// TIA Portal V20 export
// export: Created 2025-12-01T14:56:28.7894761Z, ExportSetting None, DisplayName Totally Integrated Automation Portal, DisplayVersion V20 Update 3, DisplayName TIA Portal Openness, DisplayVersion V20 Update 3, DisplayName TIA Portal Version Control Interface, DisplayVersion V20 Update 3, DisplayName STEP 7 Professional, DisplayVersion V20 Update 3, DisplayName STEP 7 Safety, DisplayVersion V20 Update 2, DisplayName WinCC Basic/Comfort/Advanced, DisplayVersion V20 Update 3, DisplayName WinCC Professional, DisplayVersion V20 Update 3, DisplayName WinCC Unified, DisplayVersion V20 Update 3
FUNCTION_BLOCK "FB415_EST_Girador_180G"   // FB415, LAD
TITLE = Control del Ramal de Salidas
{ S7_Optimized_Access := 'FALSE' }
AUTHOR : TLigero
NAME : 20160208
VERSION : 3.2
// FECHA:    27/05/2014  AUTOR: N.Rodriguez
// INSTALACION: Santomera Ampliacion 2FSS
// //////////////////////////////////
// // Registro Incidencias   ////////
// //////////////////////////////////
// FECHA:   AUTOR MODIFICACION: 
// DESCRIPCION:
// stored: AutoNumber false, SetENOAutomatically false
   VAR_INPUT
      Mesa : UInt;
      En_Tension : Bool;
      pHs_Tope : Bool;
      In_Tope_Up : Bool;
      In_Tope_Dw : Bool;
      In_Gir_Pos0 : Bool;
      In_Gir_Pos180 : Bool;
      In_Gir_Up : Bool;
      In_Gir_Dw : Bool;
      Termico_E1S3 : Bool;
      Avance_E1S3 : Bool;
      NXT_CargaOK : Bool;
      NXT_Avance : Bool;
      PRV_AVTF : Bool;
      V_TMPAus_Salida : UDInt;
      V_TMPVaciado : Time := T#10S;
      V_TOUT_Avance : Time := T#15S;
      V_TOUT_Giro_Girador : Time := T#5S;
      V_TOUT_Tope : Time := T#5S;
      V_TOUT_Elevacion_Girador : Time;
      V_TMP_Centrado : Time;
   END_VAR
   VAR_OUTPUT
      PRV_CARGA_OK : Bool;
      NXT_AVTF : Bool;
   END_VAR
   VAR
      T1_ET00 : Bool;
      T1_ET01 : Bool;
      T1_ET02 : Bool;
      T1_ET03 : Bool;
      T1_ET10 : Bool;
      T1_ET30 : Bool;
      T1_ET40 : Bool;
      T1_ET31 : Bool;
      T1_ET41 : Bool;
      T1_ET50 : Bool;
      T1_ET51 : Bool;
      MemFN_pHs : Bool;
      MemAuxFN_pHs : Bool;
      OK_Tmp_Carga : Bool;
      OK_TmpAusSalida : Bool;
      TMP_Aus_Salida : UDInt;
      TMP_En_tension : UDInt;
      TOUT_Tope { S7_SetPoint := 'True'} : TON_TIME;
      TIMVacido { S7_SetPoint := 'True'} : TON_TIME;
      TOUT_E1S3 { S7_SetPoint := 'True'} : TON_TIME;
      TOUT_Elevacion_Girador { S7_SetPoint := 'True'} : TON_TIME;
      TOUT_Giro_Girador { S7_SetPoint := 'True'} : TON_TIME;
      Tmp_Centrado { S7_SetPoint := 'True'} : TON_TIME;
   END_VAR
   VAR_TEMP
      EstadoZona : "EstadoZona";   // Estado de Zona de la Mesa
      EstadoVI : "EstadosMesa";   // Estado del Vehiculo Inteliguente de la Mesa
      ConfigFB : "UDT_ConfigFB";   // Configuracion de la FB de la Mesa
      Ok_tension : Bool;
   END_VAR
   VAR_TEMP   // added for the SCL form of the ladder/FBD networks
      _w1 : Bool;
   END_VAR
BEGIN

REGION Network 1: INICIALIZAR - Recoger las Variables de Estado de la Mesa
   // Se recoge - Estado_CBx
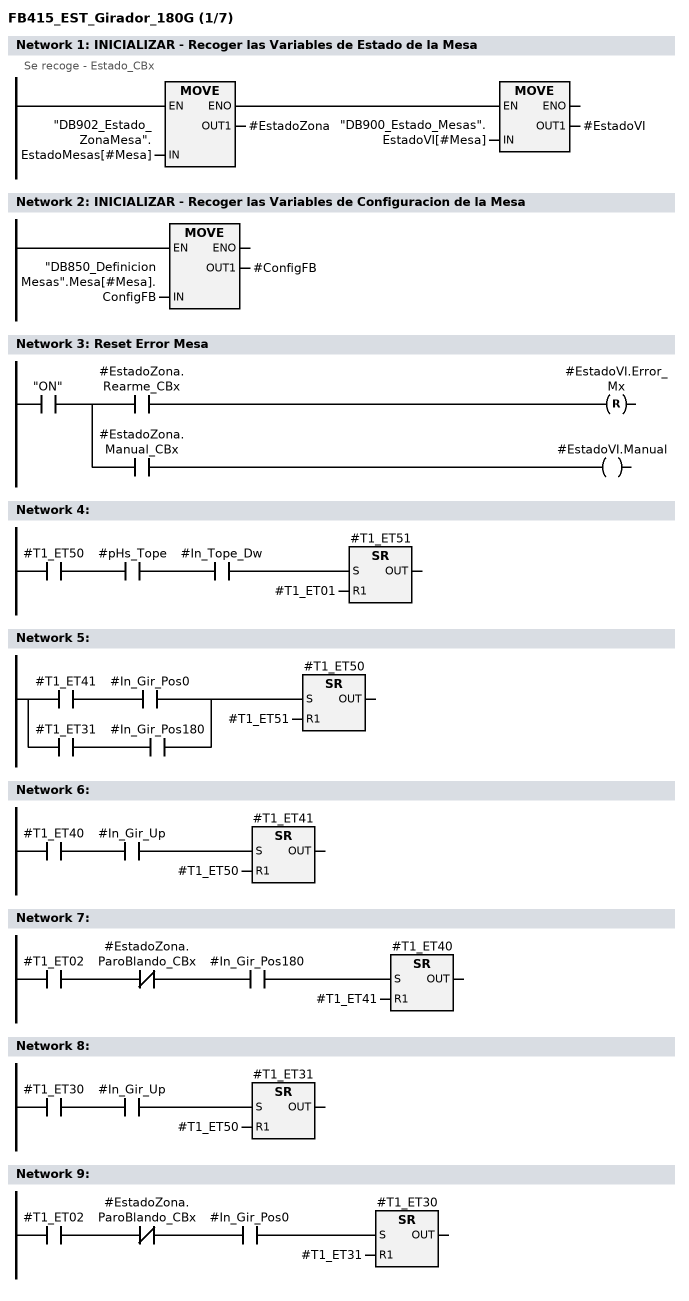
   RUNG wire#powerrail
      Move(in := "DB902_Estado_ZonaMesa".EstadoMesas[#Mesa], out1 => #EstadoZona)
      Move(in := "DB900_Estado_Mesas".EstadoVI[#Mesa], out1 => #EstadoVI)
   END_RUNG
   // the same network as SCL:
   #EstadoZona := "DB902_Estado_ZonaMesa".EstadoMesas[#Mesa];
   #EstadoVI := "DB900_Estado_Mesas".EstadoVI[#Mesa];
END_REGION

REGION Network 2: INICIALIZAR - Recoger las Variables de Configuracion de la Mesa
   RUNG wire#powerrail
      Move(in := "DB850_DefinicionMesas".Mesa[#Mesa].ConfigFB, out1 => #ConfigFB)
   END_RUNG
   // the same network as SCL:
   #ConfigFB := "DB850_DefinicionMesas".Mesa[#Mesa].ConfigFB;
END_REGION

REGION Network 3: Reset Error Mesa
   RUNG wire#powerrail
      Contact( "ON" )
      wire#w1
      Contact( #EstadoZona.Rearme_CBx )
      R_Coil( #EstadoVI.Error_Mx )
   END_RUNG
   RUNG wire#w1
      Contact( #EstadoZona.Manual_CBx )
      Coil( #EstadoVI.Manual )
   END_RUNG
   // the same network as SCL:
   IF "ON" AND #EstadoZona.Rearme_CBx THEN #EstadoVI.Error_Mx := FALSE; END_IF;
   #EstadoVI.Manual := "ON" AND #EstadoZona.Manual_CBx;
END_REGION

REGION Network 4
   RUNG wire#powerrail
      Contact( #T1_ET50 )
      Contact( #pHs_Tope )
      Contact( #In_Tope_Dw )
      S_SR(operand := #T1_ET51, r1 := #T1_ET01)
   END_RUNG
   // the same network as SCL:
   IF #T1_ET50 AND #pHs_Tope AND #In_Tope_Dw THEN
       #T1_ET51 := TRUE;   // SR flip-flop
   END_IF;
   IF #T1_ET01 THEN #T1_ET51 := FALSE; END_IF;
END_REGION

REGION Network 5
   RUNG wire#powerrail
      Contact( #T1_ET41 )
      Contact( #In_Gir_Pos0 )
      wire#w1
      S_SR(operand := #T1_ET50, r1 := #T1_ET51)
   END_RUNG
   RUNG wire#powerrail
      Contact( #T1_ET31 )
      Contact( #In_Gir_Pos180 )
   END_RUNG wire#w1
   // the same network as SCL:
   IF (#T1_ET41 AND #In_Gir_Pos0) OR (#T1_ET31 AND #In_Gir_Pos180) THEN
       #T1_ET50 := TRUE;   // SR flip-flop
   END_IF;
   IF #T1_ET51 THEN #T1_ET50 := FALSE; END_IF;
END_REGION

REGION Network 6
   RUNG wire#powerrail
      Contact( #T1_ET40 )
      Contact( #In_Gir_Up )
      S_SR(operand := #T1_ET41, r1 := #T1_ET50)
   END_RUNG
   // the same network as SCL:
   IF #T1_ET40 AND #In_Gir_Up THEN
       #T1_ET41 := TRUE;   // SR flip-flop
   END_IF;
   IF #T1_ET50 THEN #T1_ET41 := FALSE; END_IF;
END_REGION

REGION Network 7
   RUNG wire#powerrail
      Contact( #T1_ET02 )
      I_Contact( #EstadoZona.ParoBlando_CBx )
      Contact( #In_Gir_Pos180 )
      S_SR(operand := #T1_ET40, r1 := #T1_ET41)
   END_RUNG
   // the same network as SCL:
   IF #T1_ET02 AND NOT #EstadoZona.ParoBlando_CBx AND #In_Gir_Pos180 THEN
       #T1_ET40 := TRUE;   // SR flip-flop
   END_IF;
   IF #T1_ET41 THEN #T1_ET40 := FALSE; END_IF;
END_REGION

REGION Network 8
   RUNG wire#powerrail
      Contact( #T1_ET30 )
      Contact( #In_Gir_Up )
      S_SR(operand := #T1_ET31, r1 := #T1_ET50)
   END_RUNG
   // the same network as SCL:
   IF #T1_ET30 AND #In_Gir_Up THEN
       #T1_ET31 := TRUE;   // SR flip-flop
   END_IF;
   IF #T1_ET50 THEN #T1_ET31 := FALSE; END_IF;
END_REGION

REGION Network 9
   RUNG wire#powerrail
      Contact( #T1_ET02 )
      I_Contact( #EstadoZona.ParoBlando_CBx )
      Contact( #In_Gir_Pos0 )
      S_SR(operand := #T1_ET30, r1 := #T1_ET31)
   END_RUNG
   // the same network as SCL:
   IF #T1_ET02 AND NOT #EstadoZona.ParoBlando_CBx AND #In_Gir_Pos0 THEN
       #T1_ET30 := TRUE;   // SR flip-flop
   END_IF;
   IF #T1_ET31 THEN #T1_ET30 := FALSE; END_IF;
END_REGION

REGION Network 10
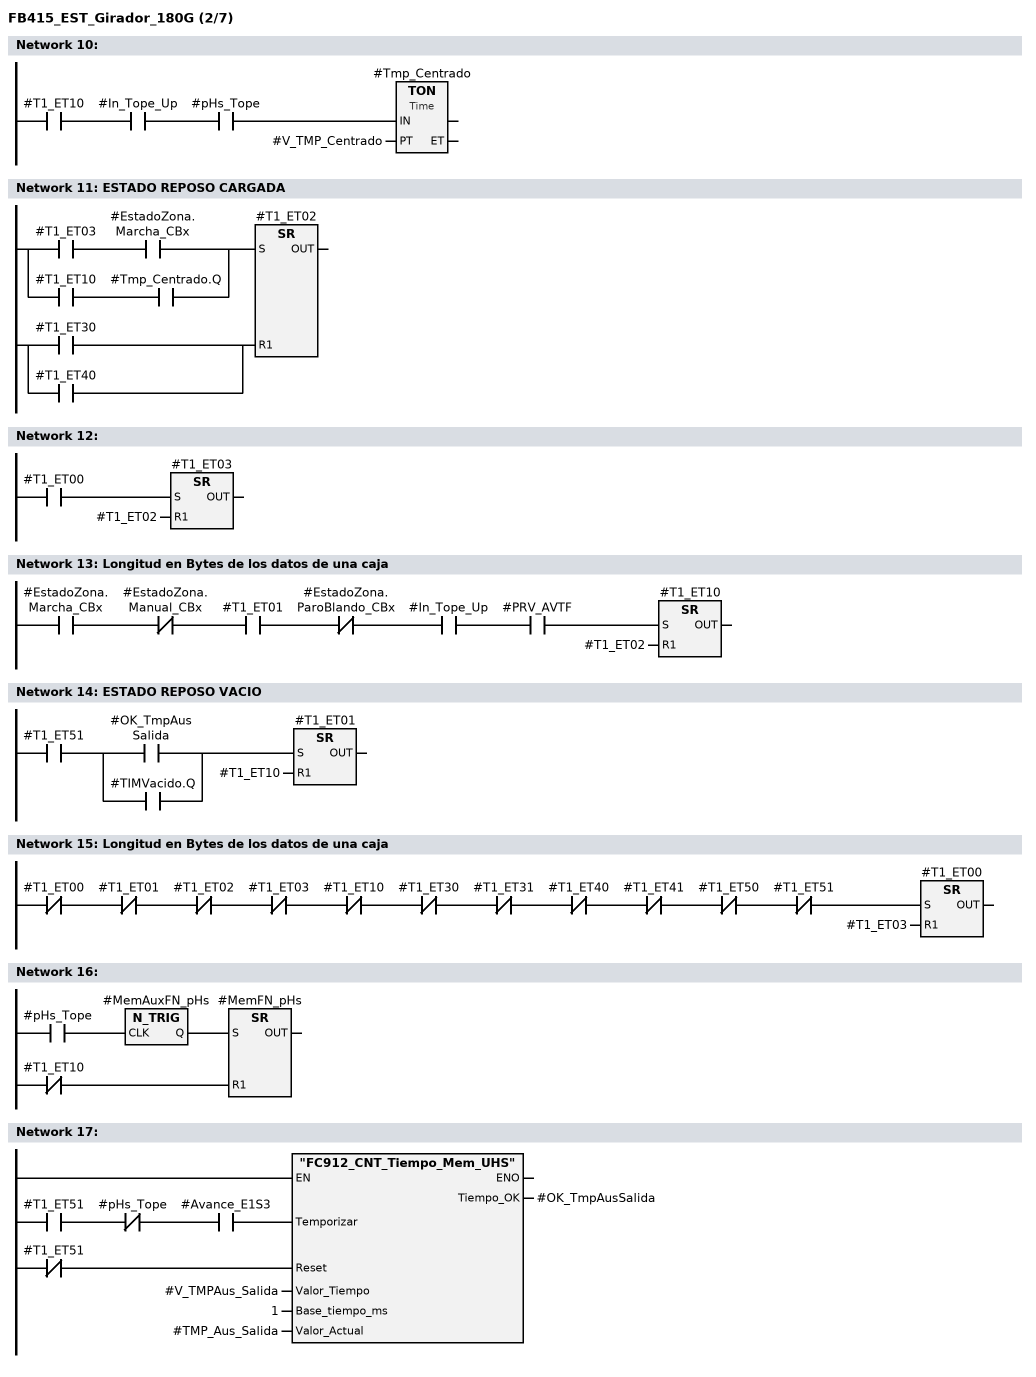
   RUNG wire#powerrail
      Contact( #T1_ET10 )
      Contact( #In_Tope_Up )
      Contact( #pHs_Tope )
      { S7_Templates := "time_type := Time" } #Tmp_Centrado.TON(pt := #V_TMP_Centrado, et =>)
   END_RUNG
   // the same network as SCL:
   #Tmp_Centrado(IN := #T1_ET10 AND #In_Tope_Up AND #pHs_Tope, PT := #V_TMP_Centrado);   // TON
END_REGION

REGION Network 11: ESTADO REPOSO CARGADA
   RUNG wire#powerrail
      Contact( #T1_ET03 )
      Contact( #EstadoZona.Marcha_CBx )
      wire#w1
      S_SR(operand := #T1_ET02, r1 := wire#w2)
   END_RUNG
   RUNG wire#powerrail
      Contact( #T1_ET10 )
      Contact( #Tmp_Centrado.Q )
   END_RUNG wire#w1
   RUNG wire#powerrail
      Contact( #T1_ET30 )
   END_RUNG wire#w2
   RUNG wire#powerrail
      Contact( #T1_ET40 )
   END_RUNG wire#w2
   // the same network as SCL:
   IF (#T1_ET03 AND #EstadoZona.Marcha_CBx) OR (#T1_ET10 AND #Tmp_Centrado.Q) THEN
       #T1_ET02 := TRUE;   // SR flip-flop
   END_IF;
   IF #T1_ET30 OR #T1_ET40 THEN #T1_ET02 := FALSE; END_IF;
END_REGION

REGION Network 12
   RUNG wire#powerrail
      Contact( #T1_ET00 )
      S_SR(operand := #T1_ET03, r1 := #T1_ET02)
   END_RUNG
   // the same network as SCL:
   IF #T1_ET00 THEN
       #T1_ET03 := TRUE;   // SR flip-flop
   END_IF;
   IF #T1_ET02 THEN #T1_ET03 := FALSE; END_IF;
END_REGION

REGION Network 13: Longitud en Bytes de los datos de una caja
   RUNG wire#powerrail
      Contact( #EstadoZona.Marcha_CBx )
      I_Contact( #EstadoZona.Manual_CBx )
      Contact( #T1_ET01 )
      I_Contact( #EstadoZona.ParoBlando_CBx )
      Contact( #In_Tope_Up )
      Contact( #PRV_AVTF )
      S_SR(operand := #T1_ET10, r1 := #T1_ET02)
   END_RUNG
   // the same network as SCL:
   IF #EstadoZona.Marcha_CBx AND NOT #EstadoZona.Manual_CBx AND #T1_ET01 AND NOT #EstadoZona.ParoBlando_CBx AND #In_Tope_Up AND #PRV_AVTF THEN
       #T1_ET10 := TRUE;   // SR flip-flop
   END_IF;
   IF #T1_ET02 THEN #T1_ET10 := FALSE; END_IF;
END_REGION

REGION Network 14: ESTADO REPOSO VACIO
   RUNG wire#powerrail
      Contact( #T1_ET51 )
      wire#w1
      Contact( #OK_TmpAusSalida )
      wire#w2
      S_SR(operand := #T1_ET01, r1 := #T1_ET10)
   END_RUNG
   RUNG wire#w1
      Contact( #TIMVacido.Q )
   END_RUNG wire#w2
   // the same network as SCL:
   IF #T1_ET51 AND (#OK_TmpAusSalida OR #TIMVacido.Q) THEN
       #T1_ET01 := TRUE;   // SR flip-flop
   END_IF;
   IF #T1_ET10 THEN #T1_ET01 := FALSE; END_IF;
END_REGION

REGION Network 15: Longitud en Bytes de los datos de una caja
   RUNG wire#powerrail
      I_Contact( #T1_ET00 )
      I_Contact( #T1_ET01 )
      I_Contact( #T1_ET02 )
      I_Contact( #T1_ET03 )
      I_Contact( #T1_ET10 )
      I_Contact( #T1_ET30 )
      I_Contact( #T1_ET31 )
      I_Contact( #T1_ET40 )
      I_Contact( #T1_ET41 )
      I_Contact( #T1_ET50 )
      I_Contact( #T1_ET51 )
      S_SR(operand := #T1_ET00, r1 := #T1_ET03)
   END_RUNG
   // the same network as SCL:
   IF NOT #T1_ET00 AND NOT #T1_ET01 AND NOT #T1_ET02 AND NOT #T1_ET03 AND NOT #T1_ET10 AND NOT #T1_ET30 AND NOT #T1_ET31 AND NOT #T1_ET40 AND NOT #T1_ET41 AND NOT #T1_ET50 AND NOT #T1_ET51 THEN
       #T1_ET00 := TRUE;   // SR flip-flop
   END_IF;
   IF #T1_ET03 THEN #T1_ET00 := FALSE; END_IF;
END_REGION

REGION Network 16
   RUNG wire#powerrail
      Contact( #pHs_Tope )
      N_Trig( #MemAuxFN_pHs )
      S_SR(operand := #MemFN_pHs, r1 := wire#w1)
   END_RUNG
   RUNG wire#powerrail
      I_Contact( #T1_ET10 )
   END_RUNG wire#w1
   // the same network as SCL:
   #_w1 := NOT #pHs_Tope AND #MemAuxFN_pHs;   // falling edge
   #MemAuxFN_pHs := #pHs_Tope;
   IF #_w1 THEN
       #MemFN_pHs := TRUE;   // SR flip-flop
   END_IF;
   IF NOT #T1_ET10 THEN #MemFN_pHs := FALSE; END_IF;
END_REGION

REGION Network 17
   RUNG wire#powerrail
      "FC912_CNT_Tiempo_Mem_UHS"(Temporizar := wire#w1, Reset := wire#w2, Valor_Tiempo := #V_TMPAus_Salida, Base_tiempo_ms := 1, Valor_Actual := #TMP_Aus_Salida, Tiempo_OK => #OK_TmpAusSalida)
   END_RUNG
   RUNG wire#powerrail
      Contact( #T1_ET51 )
      I_Contact( #pHs_Tope )
      Contact( #Avance_E1S3 )
   END_RUNG wire#w1
   RUNG wire#powerrail
      I_Contact( #T1_ET51 )
   END_RUNG wire#w2
   // the same network as SCL:
   "FC912_CNT_Tiempo_Mem_UHS"(Temporizar := #T1_ET51 AND NOT #pHs_Tope AND #Avance_E1S3,
                           Reset := NOT #T1_ET51,
                           Valor_Tiempo := #V_TMPAus_Salida,
                           Base_tiempo_ms := 1,
                           Valor_Actual := #TMP_Aus_Salida,
                           Tiempo_OK => #OK_TmpAusSalida);
END_REGION

REGION Network 18
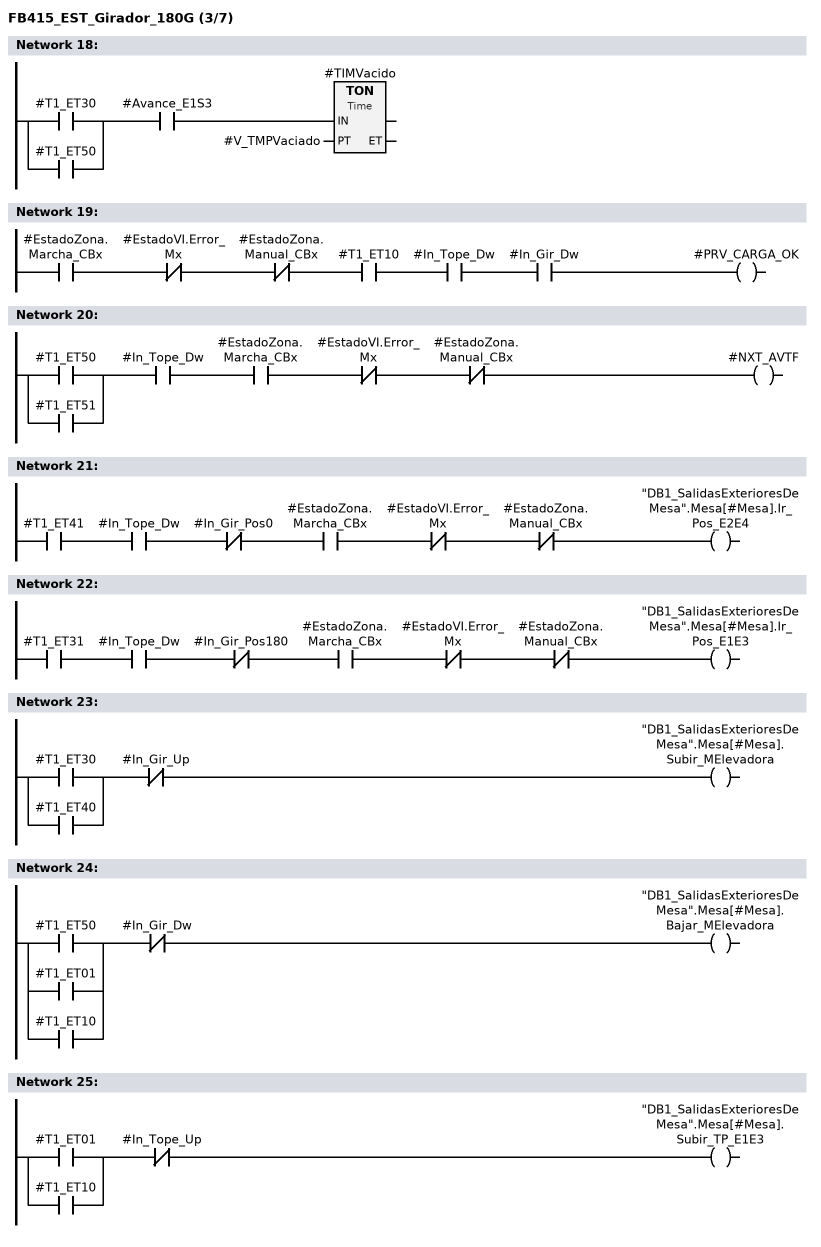
   RUNG wire#powerrail
      Contact( #T1_ET30 )
      wire#w1
      Contact( #Avance_E1S3 )
      { S7_Templates := "time_type := Time" } #TIMVacido.TON(pt := #V_TMPVaciado, et =>)
   END_RUNG
   RUNG wire#powerrail
      Contact( #T1_ET50 )
   END_RUNG wire#w1
   // the same network as SCL:
   #TIMVacido(IN := (#T1_ET30 OR #T1_ET50) AND #Avance_E1S3, PT := #V_TMPVaciado);   // TON
END_REGION

REGION Network 19
   RUNG wire#powerrail
      Contact( #EstadoZona.Marcha_CBx )
      I_Contact( #EstadoVI.Error_Mx )
      I_Contact( #EstadoZona.Manual_CBx )
      Contact( #T1_ET10 )
      Contact( #In_Tope_Dw )
      Contact( #In_Gir_Dw )
      Coil( #PRV_CARGA_OK )
   END_RUNG
   // the same network as SCL:
   #PRV_CARGA_OK := #EstadoZona.Marcha_CBx AND NOT #EstadoVI.Error_Mx AND NOT #EstadoZona.Manual_CBx AND #T1_ET10 AND #In_Tope_Dw AND #In_Gir_Dw;
END_REGION

REGION Network 20
   RUNG wire#powerrail
      Contact( #T1_ET50 )
      wire#w1
      Contact( #In_Tope_Dw )
      Contact( #EstadoZona.Marcha_CBx )
      I_Contact( #EstadoVI.Error_Mx )
      I_Contact( #EstadoZona.Manual_CBx )
      Coil( #NXT_AVTF )
   END_RUNG
   RUNG wire#powerrail
      Contact( #T1_ET51 )
   END_RUNG wire#w1
   // the same network as SCL:
   #NXT_AVTF := (#T1_ET50 OR #T1_ET51) AND #In_Tope_Dw AND #EstadoZona.Marcha_CBx AND NOT #EstadoVI.Error_Mx AND NOT #EstadoZona.Manual_CBx;
END_REGION

REGION Network 21
   RUNG wire#powerrail
      Contact( #T1_ET41 )
      Contact( #In_Tope_Dw )
      I_Contact( #In_Gir_Pos0 )
      Contact( #EstadoZona.Marcha_CBx )
      I_Contact( #EstadoVI.Error_Mx )
      I_Contact( #EstadoZona.Manual_CBx )
      Coil( "DB1_SalidasExterioresDeMesa".Mesa[#Mesa].Ir_Pos_E2E4 )
   END_RUNG
   // the same network as SCL:
   "DB1_SalidasExterioresDeMesa".Mesa[#Mesa].Ir_Pos_E2E4 := #T1_ET41 AND #In_Tope_Dw AND NOT #In_Gir_Pos0 AND #EstadoZona.Marcha_CBx AND NOT #EstadoVI.Error_Mx AND NOT #EstadoZona.Manual_CBx;
END_REGION

REGION Network 22
   RUNG wire#powerrail
      Contact( #T1_ET31 )
      Contact( #In_Tope_Dw )
      I_Contact( #In_Gir_Pos180 )
      Contact( #EstadoZona.Marcha_CBx )
      I_Contact( #EstadoVI.Error_Mx )
      I_Contact( #EstadoZona.Manual_CBx )
      Coil( "DB1_SalidasExterioresDeMesa".Mesa[#Mesa].Ir_Pos_E1E3 )
   END_RUNG
   // the same network as SCL:
   "DB1_SalidasExterioresDeMesa".Mesa[#Mesa].Ir_Pos_E1E3 := #T1_ET31 AND #In_Tope_Dw AND NOT #In_Gir_Pos180 AND #EstadoZona.Marcha_CBx AND NOT #EstadoVI.Error_Mx AND NOT #EstadoZona.Manual_CBx;
END_REGION

REGION Network 23
   RUNG wire#powerrail
      Contact( #T1_ET30 )
      wire#w1
      I_Contact( #In_Gir_Up )
      Coil( "DB1_SalidasExterioresDeMesa".Mesa[#Mesa].Subir_MElevadora )
   END_RUNG
   RUNG wire#powerrail
      Contact( #T1_ET40 )
   END_RUNG wire#w1
   // the same network as SCL:
   "DB1_SalidasExterioresDeMesa".Mesa[#Mesa].Subir_MElevadora := (#T1_ET30 OR #T1_ET40) AND NOT #In_Gir_Up;
END_REGION

REGION Network 24
   RUNG wire#powerrail
      Contact( #T1_ET50 )
      wire#w1
      I_Contact( #In_Gir_Dw )
      Coil( "DB1_SalidasExterioresDeMesa".Mesa[#Mesa].Bajar_MElevadora )
   END_RUNG
   RUNG wire#powerrail
      Contact( #T1_ET01 )
   END_RUNG wire#w1
   RUNG wire#powerrail
      Contact( #T1_ET10 )
   END_RUNG wire#w1
   // the same network as SCL:
   "DB1_SalidasExterioresDeMesa".Mesa[#Mesa].Bajar_MElevadora := (#T1_ET50 OR #T1_ET01 OR #T1_ET10) AND NOT #In_Gir_Dw;
END_REGION

REGION Network 25
   RUNG wire#powerrail
      Contact( #T1_ET01 )
      wire#w1
      I_Contact( #In_Tope_Up )
      Coil( "DB1_SalidasExterioresDeMesa".Mesa[#Mesa].Subir_TP_E1E3 )
   END_RUNG
   RUNG wire#powerrail
      Contact( #T1_ET10 )
   END_RUNG wire#w1
   // the same network as SCL:
   "DB1_SalidasExterioresDeMesa".Mesa[#Mesa].Subir_TP_E1E3 := (#T1_ET01 OR #T1_ET10) AND NOT #In_Tope_Up;
END_REGION

REGION Network 26
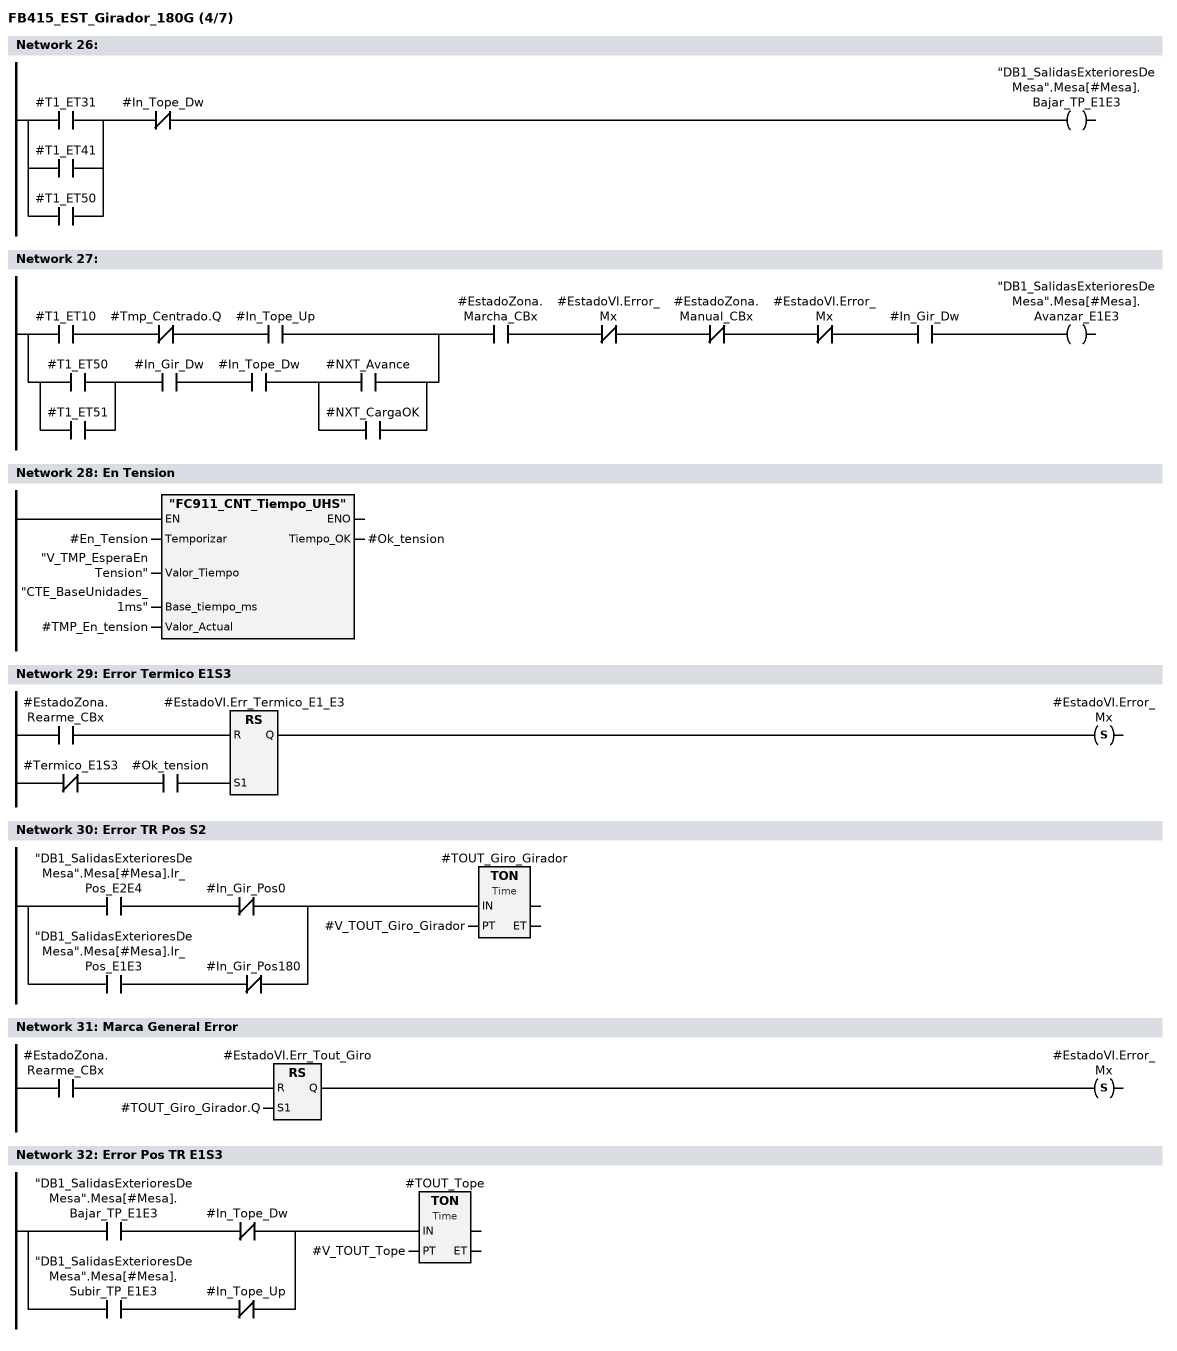
   RUNG wire#powerrail
      Contact( #T1_ET31 )
      wire#w1
      I_Contact( #In_Tope_Dw )
      Coil( "DB1_SalidasExterioresDeMesa".Mesa[#Mesa].Bajar_TP_E1E3 )
   END_RUNG
   RUNG wire#powerrail
      Contact( #T1_ET41 )
   END_RUNG wire#w1
   RUNG wire#powerrail
      Contact( #T1_ET50 )
   END_RUNG wire#w1
   // the same network as SCL:
   "DB1_SalidasExterioresDeMesa".Mesa[#Mesa].Bajar_TP_E1E3 := (#T1_ET31 OR #T1_ET41 OR #T1_ET50) AND NOT #In_Tope_Dw;
END_REGION

REGION Network 27
   RUNG wire#powerrail
      Contact( #T1_ET10 )
      I_Contact( #Tmp_Centrado.Q )
      Contact( #In_Tope_Up )
      wire#w1
      Contact( #EstadoZona.Marcha_CBx )
      I_Contact( #EstadoVI.Error_Mx )
      I_Contact( #EstadoZona.Manual_CBx )
      I_Contact( #EstadoVI.Error_Mx )
      Contact( #In_Gir_Dw )
      Coil( "DB1_SalidasExterioresDeMesa".Mesa[#Mesa].Avanzar_E1E3 )
   END_RUNG
   RUNG wire#powerrail
      Contact( #T1_ET50 )
      wire#w2
      Contact( #In_Gir_Dw )
      Contact( #In_Tope_Dw )
      wire#w3
      Contact( #NXT_Avance )
   END_RUNG wire#w1
   RUNG wire#powerrail
      Contact( #T1_ET51 )
   END_RUNG wire#w2
   RUNG wire#w3
      Contact( #NXT_CargaOK )
   END_RUNG wire#w1
   // the same network as SCL:
   "DB1_SalidasExterioresDeMesa".Mesa[#Mesa].Avanzar_E1E3 := ((#T1_ET10 AND NOT #Tmp_Centrado.Q AND #In_Tope_Up) OR ((#T1_ET50 OR #T1_ET51) AND #In_Gir_Dw AND #In_Tope_Dw AND (#NXT_Avance OR #NXT_CargaOK))) AND #EstadoZona.Marcha_CBx AND NOT #EstadoVI.Error_Mx AND NOT #EstadoZona.Manual_CBx AND NOT #EstadoVI.Error_Mx AND #In_Gir_Dw;
END_REGION

REGION Network 28: En Tension
   RUNG wire#powerrail
      "FC911_CNT_Tiempo_UHS"(Temporizar := #En_Tension, Valor_Tiempo := "V_TMP_EsperaEnTension", Base_tiempo_ms := "CTE_BaseUnidades_1ms", Valor_Actual := #TMP_En_tension, Tiempo_OK => #Ok_tension)
   END_RUNG
   // the same network as SCL:
   "FC911_CNT_Tiempo_UHS"(Temporizar := #En_Tension,
                          Valor_Tiempo := "V_TMP_EsperaEnTension",
                          Base_tiempo_ms := "CTE_BaseUnidades_1ms",
                          Valor_Actual := #TMP_En_tension,
                          Tiempo_OK => #Ok_tension);
END_REGION

REGION Network 29: Error Termico E1S3
   RUNG wire#powerrail
      Contact( #EstadoZona.Rearme_CBx )
      S_RS(operand := #EstadoVI.Err_Termico_E1_E3, s1 := wire#w1)
      S_Coil( #EstadoVI.Error_Mx )
   END_RUNG
   RUNG wire#powerrail
      I_Contact( #Termico_E1S3 )
      Contact( #Ok_tension )
   END_RUNG wire#w1
   // the same network as SCL:
   IF #EstadoZona.Rearme_CBx THEN
       #EstadoVI.Err_Termico_E1_E3 := FALSE;   // RS flip-flop
   END_IF;
   IF NOT #Termico_E1S3 AND #Ok_tension THEN #EstadoVI.Err_Termico_E1_E3 := TRUE; END_IF;
   IF #EstadoVI.Err_Termico_E1_E3 THEN #EstadoVI.Error_Mx := TRUE; END_IF;
END_REGION

REGION Network 30: Error TR Pos S2
   RUNG wire#powerrail
      Contact( "DB1_SalidasExterioresDeMesa".Mesa[#Mesa].Ir_Pos_E2E4 )
      I_Contact( #In_Gir_Pos0 )
      wire#w1
      { S7_Templates := "time_type := Time" } #TOUT_Giro_Girador.TON(pt := #V_TOUT_Giro_Girador, et =>)
   END_RUNG
   RUNG wire#powerrail
      Contact( "DB1_SalidasExterioresDeMesa".Mesa[#Mesa].Ir_Pos_E1E3 )
      I_Contact( #In_Gir_Pos180 )
   END_RUNG wire#w1
   // the same network as SCL:
   #TOUT_Giro_Girador(IN := ("DB1_SalidasExterioresDeMesa".Mesa[#Mesa].Ir_Pos_E2E4 AND NOT #In_Gir_Pos0) OR ("DB1_SalidasExterioresDeMesa".Mesa[#Mesa].Ir_Pos_E1E3 AND NOT #In_Gir_Pos180),   // TON
                      PT := #V_TOUT_Giro_Girador);
END_REGION

REGION Network 31: Marca General Error
   RUNG wire#powerrail
      Contact( #EstadoZona.Rearme_CBx )
      S_RS(operand := #EstadoVI.Err_Tout_Giro, s1 := #TOUT_Giro_Girador.Q)
      S_Coil( #EstadoVI.Error_Mx )
   END_RUNG
   // the same network as SCL:
   IF #EstadoZona.Rearme_CBx THEN
       #EstadoVI.Err_Tout_Giro := FALSE;   // RS flip-flop
   END_IF;
   IF #TOUT_Giro_Girador.Q THEN #EstadoVI.Err_Tout_Giro := TRUE; END_IF;
   IF #EstadoVI.Err_Tout_Giro THEN #EstadoVI.Error_Mx := TRUE; END_IF;
END_REGION

REGION Network 32: Error Pos TR E1S3
   RUNG wire#powerrail
      Contact( "DB1_SalidasExterioresDeMesa".Mesa[#Mesa].Bajar_TP_E1E3 )
      I_Contact( #In_Tope_Dw )
      wire#w1
      { S7_Templates := "time_type := Time" } #TOUT_Tope.TON(pt := #V_TOUT_Tope, et =>)
   END_RUNG
   RUNG wire#powerrail
      Contact( "DB1_SalidasExterioresDeMesa".Mesa[#Mesa].Subir_TP_E1E3 )
      I_Contact( #In_Tope_Up )
   END_RUNG wire#w1
   // the same network as SCL:
   #TOUT_Tope(IN := ("DB1_SalidasExterioresDeMesa".Mesa[#Mesa].Bajar_TP_E1E3 AND NOT #In_Tope_Dw) OR ("DB1_SalidasExterioresDeMesa".Mesa[#Mesa].Subir_TP_E1E3 AND NOT #In_Tope_Up),   // TON
              PT := #V_TOUT_Tope);
END_REGION

REGION Network 33: Marca General Error
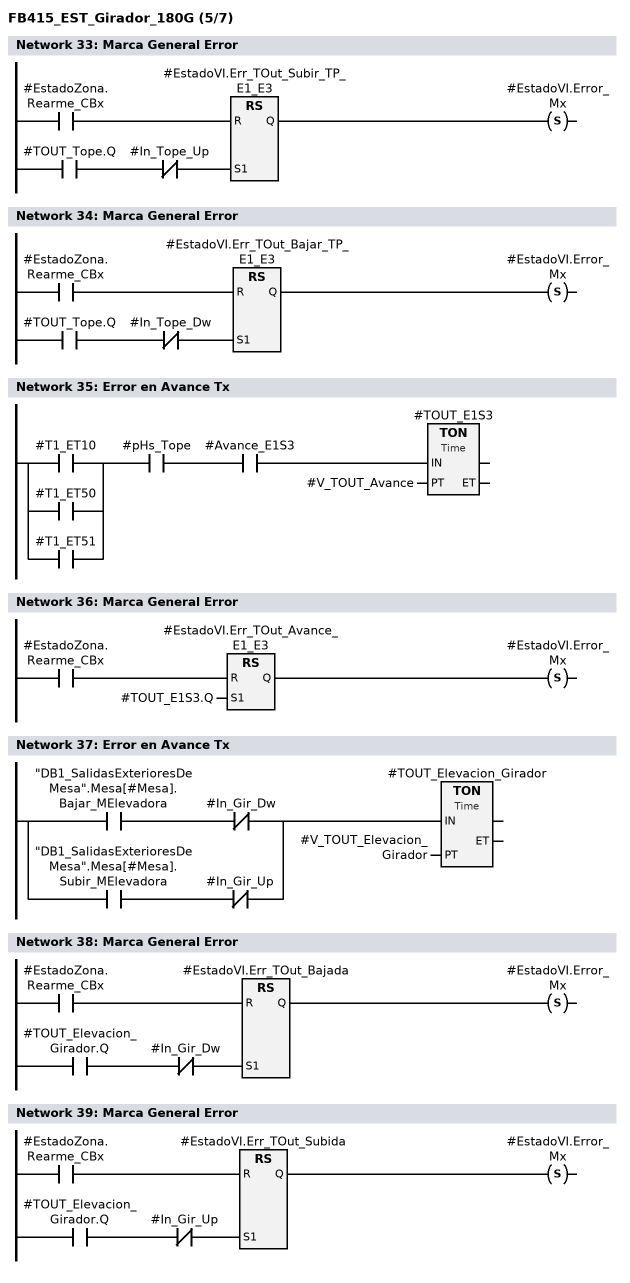
   RUNG wire#powerrail
      Contact( #EstadoZona.Rearme_CBx )
      S_RS(operand := #EstadoVI.Err_TOut_Subir_TP_E1_E3, s1 := wire#w1)
      S_Coil( #EstadoVI.Error_Mx )
   END_RUNG
   RUNG wire#powerrail
      Contact( #TOUT_Tope.Q )
      I_Contact( #In_Tope_Up )
   END_RUNG wire#w1
   // the same network as SCL:
   IF #EstadoZona.Rearme_CBx THEN
       #EstadoVI.Err_TOut_Subir_TP_E1_E3 := FALSE;   // RS flip-flop
   END_IF;
   IF #TOUT_Tope.Q AND NOT #In_Tope_Up THEN #EstadoVI.Err_TOut_Subir_TP_E1_E3 := TRUE; END_IF;
   IF #EstadoVI.Err_TOut_Subir_TP_E1_E3 THEN #EstadoVI.Error_Mx := TRUE; END_IF;
END_REGION

REGION Network 34: Marca General Error
   RUNG wire#powerrail
      Contact( #EstadoZona.Rearme_CBx )
      S_RS(operand := #EstadoVI.Err_TOut_Bajar_TP_E1_E3, s1 := wire#w1)
      S_Coil( #EstadoVI.Error_Mx )
   END_RUNG
   RUNG wire#powerrail
      Contact( #TOUT_Tope.Q )
      I_Contact( #In_Tope_Dw )
   END_RUNG wire#w1
   // the same network as SCL:
   IF #EstadoZona.Rearme_CBx THEN
       #EstadoVI.Err_TOut_Bajar_TP_E1_E3 := FALSE;   // RS flip-flop
   END_IF;
   IF #TOUT_Tope.Q AND NOT #In_Tope_Dw THEN #EstadoVI.Err_TOut_Bajar_TP_E1_E3 := TRUE; END_IF;
   IF #EstadoVI.Err_TOut_Bajar_TP_E1_E3 THEN #EstadoVI.Error_Mx := TRUE; END_IF;
END_REGION

REGION Network 35: Error en Avance Tx
   RUNG wire#powerrail
      Contact( #T1_ET10 )
      wire#w1
      Contact( #pHs_Tope )
      Contact( #Avance_E1S3 )
      { S7_Templates := "time_type := Time" } #TOUT_E1S3.TON(pt := #V_TOUT_Avance, et =>)
   END_RUNG
   RUNG wire#powerrail
      Contact( #T1_ET50 )
   END_RUNG wire#w1
   RUNG wire#powerrail
      Contact( #T1_ET51 )
   END_RUNG wire#w1
   // the same network as SCL:
   #TOUT_E1S3(IN := (#T1_ET10 OR #T1_ET50 OR #T1_ET51) AND #pHs_Tope AND #Avance_E1S3, PT := #V_TOUT_Avance);   // TON
END_REGION

REGION Network 36: Marca General Error
   RUNG wire#powerrail
      Contact( #EstadoZona.Rearme_CBx )
      S_RS(operand := #EstadoVI.Err_TOut_Avance_E1_E3, s1 := #TOUT_E1S3.Q)
      S_Coil( #EstadoVI.Error_Mx )
   END_RUNG
   // the same network as SCL:
   IF #EstadoZona.Rearme_CBx THEN
       #EstadoVI.Err_TOut_Avance_E1_E3 := FALSE;   // RS flip-flop
   END_IF;
   IF #TOUT_E1S3.Q THEN #EstadoVI.Err_TOut_Avance_E1_E3 := TRUE; END_IF;
   IF #EstadoVI.Err_TOut_Avance_E1_E3 THEN #EstadoVI.Error_Mx := TRUE; END_IF;
END_REGION

REGION Network 37: Error en Avance Tx
   RUNG wire#powerrail
      Contact( "DB1_SalidasExterioresDeMesa".Mesa[#Mesa].Bajar_MElevadora )
      I_Contact( #In_Gir_Dw )
      wire#w1
      { S7_Templates := "time_type := Time" } #TOUT_Elevacion_Girador.TON(pt := #V_TOUT_Elevacion_Girador, et =>)
   END_RUNG
   RUNG wire#powerrail
      Contact( "DB1_SalidasExterioresDeMesa".Mesa[#Mesa].Subir_MElevadora )
      I_Contact( #In_Gir_Up )
   END_RUNG wire#w1
   // the same network as SCL:
   #TOUT_Elevacion_Girador(IN := ("DB1_SalidasExterioresDeMesa".Mesa[#Mesa].Bajar_MElevadora AND NOT #In_Gir_Dw) OR ("DB1_SalidasExterioresDeMesa".Mesa[#Mesa].Subir_MElevadora AND NOT #In_Gir_Up),   // TON
                           PT := #V_TOUT_Elevacion_Girador);
END_REGION

REGION Network 38: Marca General Error
   RUNG wire#powerrail
      Contact( #EstadoZona.Rearme_CBx )
      S_RS(operand := #EstadoVI.Err_TOut_Bajada, s1 := wire#w1)
      S_Coil( #EstadoVI.Error_Mx )
   END_RUNG
   RUNG wire#powerrail
      Contact( #TOUT_Elevacion_Girador.Q )
      I_Contact( #In_Gir_Dw )
   END_RUNG wire#w1
   // the same network as SCL:
   IF #EstadoZona.Rearme_CBx THEN
       #EstadoVI.Err_TOut_Bajada := FALSE;   // RS flip-flop
   END_IF;
   IF #TOUT_Elevacion_Girador.Q AND NOT #In_Gir_Dw THEN #EstadoVI.Err_TOut_Bajada := TRUE; END_IF;
   IF #EstadoVI.Err_TOut_Bajada THEN #EstadoVI.Error_Mx := TRUE; END_IF;
END_REGION

REGION Network 39: Marca General Error
   RUNG wire#powerrail
      Contact( #EstadoZona.Rearme_CBx )
      S_RS(operand := #EstadoVI.Err_TOut_Subida, s1 := wire#w1)
      S_Coil( #EstadoVI.Error_Mx )
   END_RUNG
   RUNG wire#powerrail
      Contact( #TOUT_Elevacion_Girador.Q )
      I_Contact( #In_Gir_Up )
   END_RUNG wire#w1
   // the same network as SCL:
   IF #EstadoZona.Rearme_CBx THEN
       #EstadoVI.Err_TOut_Subida := FALSE;   // RS flip-flop
   END_IF;
   IF #TOUT_Elevacion_Girador.Q AND NOT #In_Gir_Up THEN #EstadoVI.Err_TOut_Subida := TRUE; END_IF;
   IF #EstadoVI.Err_TOut_Subida THEN #EstadoVI.Error_Mx := TRUE; END_IF;
END_REGION

REGION Network 40: ESTADOS MESA 1
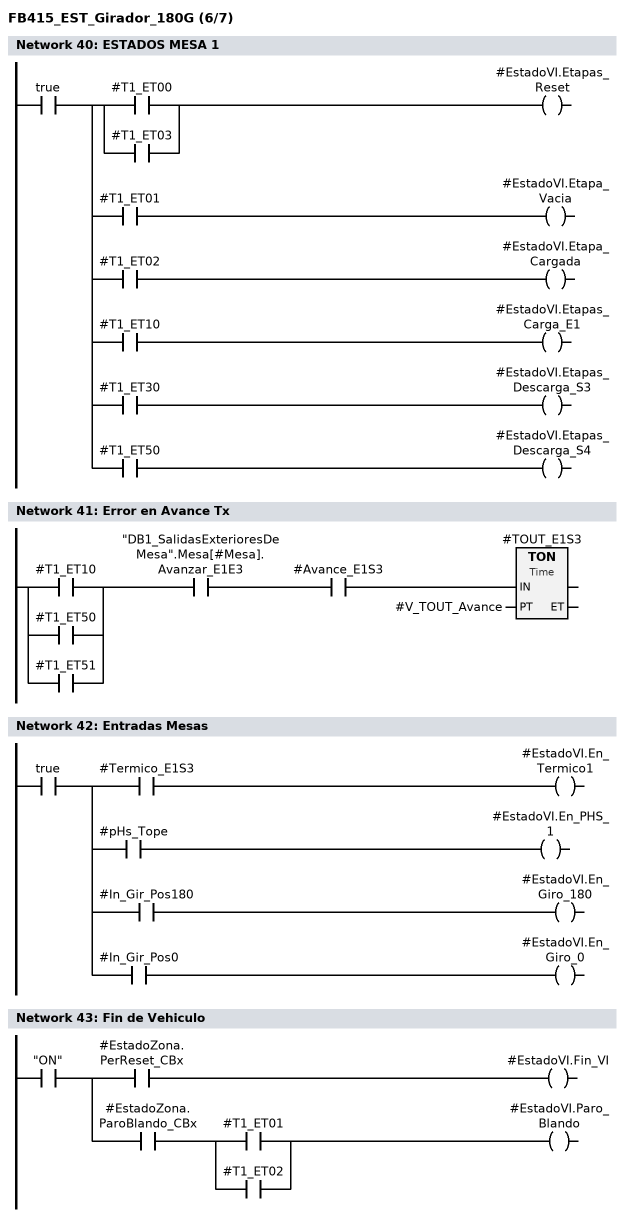
   RUNG wire#powerrail
      Contact( true )
      wire#w1
      Contact( #T1_ET00 )
      wire#w2
      Coil( #EstadoVI.Etapas_Reset )
   END_RUNG
   RUNG wire#w1
      Contact( #T1_ET03 )
   END_RUNG wire#w2
   RUNG wire#w1
      Contact( #T1_ET01 )
      Coil( #EstadoVI.Etapa_Vacia )
   END_RUNG
   RUNG wire#w1
      Contact( #T1_ET02 )
      Coil( #EstadoVI.Etapa_Cargada )
   END_RUNG
   RUNG wire#w1
      Contact( #T1_ET10 )
      Coil( #EstadoVI.Etapas_Carga_E1 )
   END_RUNG
   RUNG wire#w1
      Contact( #T1_ET30 )
      Coil( #EstadoVI.Etapas_Descarga_S3 )
   END_RUNG
   RUNG wire#w1
      Contact( #T1_ET50 )
      Coil( #EstadoVI.Etapas_Descarga_S4 )
   END_RUNG
   // the same network as SCL:
   #EstadoVI.Etapas_Reset := true AND (#T1_ET00 OR #T1_ET03);
   #EstadoVI.Etapa_Vacia := true AND #T1_ET01;
   #EstadoVI.Etapa_Cargada := true AND #T1_ET02;
   #EstadoVI.Etapas_Carga_E1 := true AND #T1_ET10;
   #EstadoVI.Etapas_Descarga_S3 := true AND #T1_ET30;
   #EstadoVI.Etapas_Descarga_S4 := true AND #T1_ET50;
END_REGION

REGION Network 41: Error en Avance Tx
   RUNG wire#powerrail
      Contact( #T1_ET10 )
      wire#w1
      Contact( "DB1_SalidasExterioresDeMesa".Mesa[#Mesa].Avanzar_E1E3 )
      Contact( #Avance_E1S3 )
      { S7_Templates := "time_type := Time" } #TOUT_E1S3.TON(pt := #V_TOUT_Avance, et =>)
   END_RUNG
   RUNG wire#powerrail
      Contact( #T1_ET50 )
   END_RUNG wire#w1
   RUNG wire#powerrail
      Contact( #T1_ET51 )
   END_RUNG wire#w1
   // the same network as SCL:
   #TOUT_E1S3(IN := (#T1_ET10 OR #T1_ET50 OR #T1_ET51) AND "DB1_SalidasExterioresDeMesa".Mesa[#Mesa].Avanzar_E1E3 AND #Avance_E1S3,   // TON
              PT := #V_TOUT_Avance);
END_REGION

REGION Network 42: Entradas Mesas
   RUNG wire#powerrail
      Contact( true )
      wire#w1
      Contact( #Termico_E1S3 )
      Coil( #EstadoVI.En_Termico1 )
   END_RUNG
   RUNG wire#w1
      Contact( #pHs_Tope )
      Coil( #EstadoVI.En_PHS_1 )
   END_RUNG
   RUNG wire#w1
      Contact( #In_Gir_Pos180 )
      Coil( #EstadoVI.En_Giro_180 )
   END_RUNG
   RUNG wire#w1
      Contact( #In_Gir_Pos0 )
      Coil( #EstadoVI.En_Giro_0 )
   END_RUNG
   // the same network as SCL:
   #EstadoVI.En_Termico1 := true AND #Termico_E1S3;
   #EstadoVI.En_PHS_1 := true AND #pHs_Tope;
   #EstadoVI.En_Giro_180 := true AND #In_Gir_Pos180;
   #EstadoVI.En_Giro_0 := true AND #In_Gir_Pos0;
END_REGION

REGION Network 43: Fin de Vehiculo
   RUNG wire#powerrail
      Contact( "ON" )
      wire#w1
      Contact( #EstadoZona.PerReset_CBx )
      Coil( #EstadoVI.Fin_VI )
   END_RUNG
   RUNG wire#w1
      Contact( #EstadoZona.ParoBlando_CBx )
      wire#w2
      Contact( #T1_ET01 )
      wire#w3
      Coil( #EstadoVI.Paro_Blando )
   END_RUNG
   RUNG wire#w2
      Contact( #T1_ET02 )
   END_RUNG wire#w3
   // the same network as SCL:
   #EstadoVI.Fin_VI := "ON" AND #EstadoZona.PerReset_CBx;
   #EstadoVI.Paro_Blando := "ON" AND #EstadoZona.ParoBlando_CBx AND (#T1_ET01 OR #T1_ET02);
END_REGION

REGION Network 44: Salidas Mesas
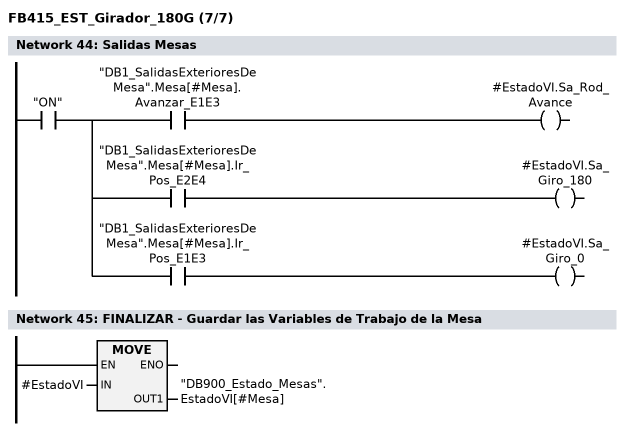
   RUNG wire#powerrail
      Contact( "ON" )
      wire#w1
      Contact( "DB1_SalidasExterioresDeMesa".Mesa[#Mesa].Avanzar_E1E3 )
      Coil( #EstadoVI.Sa_Rod_Avance )
   END_RUNG
   RUNG wire#w1
      Contact( "DB1_SalidasExterioresDeMesa".Mesa[#Mesa].Ir_Pos_E2E4 )
      Coil( #EstadoVI.Sa_Giro_180 )
   END_RUNG
   RUNG wire#w1
      Contact( "DB1_SalidasExterioresDeMesa".Mesa[#Mesa].Ir_Pos_E1E3 )
      Coil( #EstadoVI.Sa_Giro_0 )
   END_RUNG
   // the same network as SCL:
   #EstadoVI.Sa_Rod_Avance := "ON" AND "DB1_SalidasExterioresDeMesa".Mesa[#Mesa].Avanzar_E1E3;
   #EstadoVI.Sa_Giro_180 := "ON" AND "DB1_SalidasExterioresDeMesa".Mesa[#Mesa].Ir_Pos_E2E4;
   #EstadoVI.Sa_Giro_0 := "ON" AND "DB1_SalidasExterioresDeMesa".Mesa[#Mesa].Ir_Pos_E1E3;
END_REGION

REGION Network 45: FINALIZAR - Guardar las Variables de Trabajo de la Mesa
   RUNG wire#powerrail
      Move(in := #EstadoVI, out1 => "DB900_Estado_Mesas".EstadoVI[#Mesa])
   END_RUNG
   // the same network as SCL:
   "DB900_Estado_Mesas".EstadoVI[#Mesa] := #EstadoVI;
END_REGION
END_FUNCTION_BLOCK
